TYPE ST_Initialisierungsroutine :
STRUCT

    MGMT_Parameter : ST_FB_MGMT_Parameter;
	Netze_Parameter :ST_Netze_Parameter;

	Anlage_BSp_Parameter	: ST_BSp_Parameter;
	Anlage_Bel_Parameter	: ST_Bel_Parameter;
	Anlage_BHKW_921_Parameter	: ST_BHKW_Parameter;
	Anlage_BHKW_922_Parameter	: ST_BHKW_Parameter;
	Anlage_BWK_Parameter	: ST_BWK_Parameter;
	Anlage_DLK_Parameter	: ST_DLK_Parameter;
	Anlage_HES_Parameter	: ST_HES_Parameter;
	Anlage_HO_Parameter		: ST_HO_Parameter;
	Anlage_LA_Parameter		: ST_LA_Parameter;
	Anlage_MVHW_Parameter	: ST_MV_JAVA_Parameter;
	Anlage_MVKW_Parameter	: ST_MV_MAFAC_GT_Parameter;
	Anlage_WP_946_Parameter		: ST_WP_Parameter;

	System_AFA_Parameter	: ST_System_AFA_Parameter;
	System_AKM_Parameter	: ST_System_AKM_Parameter;
	System_Bel_Parameter	: ST_System_Bel_Parameter;
	System_BHKW_Parameter	: ST_System_BHKW_Parameter;
	System_BSp_Parameter	: ST_System_BSp_Parameter;
	System_BSp_KueW_Parameter	: ST_System_BSp_KueW_Parameter;
	System_BSp_Verb_Parameter	: ST_System_BSp_Verb_Parameter;
	System_BWK_Parameter	: ST_System_BWK_Parameter;
	System_DLK_Parameter	: ST_System_DLK_Parameter;
	System_FBT_Parameter	: ST_System_FBT_Parameter;
	System_HES_Parameter	: ST_System_HES_Parameter;
	System_HOHW_Parameter	: ST_System_HOHW_Parameter;
	System_HOWW_Parameter	: ST_System_HOWW_Parameter;
	System_HS_Parameter		: ST_System_HS_Parameter;
	System_KKKW_Parameter	: ST_System_KKKW_Parameter;
	System_MVWW_Parameter	: ST_System_MVWW_Parameter;
	System_LA_Parameter		: ST_System_LA_Parameter;
	System_MVHW_Parameter	: ST_System_MVHW_Parameter;
	System_MVKW_Parameter	: ST_System_MVKW_Parameter;
	System_SHZ_Parameter	: ST_System_SHZ_Parameter;
	System_ThNTZ_Parameter	: ST_ThNTZ_Parameter;
	System_WDT_Parameter	: ST_System_WDT_Parameter;
	System_WT_HWW_Parameter	: ST_System_WT_HWW_Parameter;
	System_WP_946_Parameter		: ST_System_WP_Parameter;

	Fenster_Halle_OST_Parameter		: ST_Fenster_Parameter;
	Fenster_Halle_WEST_Parameter	: ST_Fenster_Parameter;


	Stellventil_100_Parameter	: ST_SV_Parameter;
	Stellventil_105_Parameter	:  ST_SV_Parameter;
	Stellventil_145_Parameter	:  ST_SV_Parameter;
	Stellventil_191_Parameter	: ST_SV_Parameter;
	Stellventil_205_Parameter	:  ST_SV_Parameter;
	Stellventil_215_Parameter	:  ST_SV_Parameter;
	Stellventil_235_Parameter	:  ST_SV_Parameter;
	Stellventil_245_Parameter	:  ST_SV_Parameter;
	Stellventil_251_Parameter	: ST_SV_Parameter;
	Stellventil_261_Parameter	: ST_SV_Parameter;
	Stellventil_300_Parameter	:  ST_SV_Parameter;
	Stellventil_315_Parameter	:  ST_SV_Parameter;
	Stellventil_321_Parameter	:  ST_SV_Parameter;
	Stellventil_322_Parameter	:  ST_SV_Parameter;
	Stellventil_331_Parameter	:  ST_SV_Parameter;
	Stellventil_361_Parameter	:  ST_SV_Parameter;
	Stellventil_423_Parameter	:  ST_SV_Parameter;
	Stellventil_424_Parameter	: ST_SV_Parameter;
	Stellventil_453_Parameter	: ST_SV_Parameter;
	Stellventil_454_Parameter	: ST_SV_Parameter;
	Stellventil_401_402_Parameter	: ST_SV_Parameter;
	Stellventil_403_404_Parameter	: ST_SV_Parameter;
	Stellventil_504_505_Parameter	:  ST_SV_Parameter;
	Stellventil_605_Parameter	: ST_SV_Parameter;

	Stellventil_146_Parameter	: ST_SV_Parameter;
	Stellventil_246_Parameter	:  ST_SV_Parameter;

	Pumpe_100_Parameter			: ST_PU_Parameter;
	Pumpe_105_Parameter			: ST_PU_Parameter;
	Pumpe_145_Parameter			: ST_PU_Parameter;
	Pumpe_191_Parameter			: ST_PU_Parameter;
	Pumpe_205_Parameter			: ST_PU_Parameter;
	Pumpe_215_Parameter			: ST_PU_Parameter;
	Pumpe_235_Parameter			: ST_PU_Parameter;
	Pumpe_245_Parameter			: ST_PU_Parameter;
	Pumpe_251_Parameter			: ST_PU_Parameter;
	Pumpe_261_Parameter			: ST_PU_Parameter;
	Pumpe_300_Parameter			: ST_PU_Parameter;
	Pumpe_315_Parameter			: ST_PU_Parameter;
	Pumpe_321_Parameter			: ST_PU_Parameter;
	Pumpe_322_Parameter			: ST_PU_Parameter;
	Pumpe_350_Parameter			: ST_PU_Parameter;
	Pumpe_361_Parameter			: ST_PU_Parameter;
	Pumpe_405_Parameter			: ST_PU_Parameter;
	Pumpe_425_Parameter			: ST_PU_Parameter;
	Pumpe_500_Parameter			: ST_PU_Parameter;
	Pumpe_600_Parameter			: ST_PU_Parameter;
	Pumpe_690_Parameter			: ST_PU_Schuetz_Parameter;
	Pumpe_710_Parameter			: ST_PU_Schuetz_Parameter;
	Pumpe_716_Parameter			: ST_PU_Schuetz_Parameter;
	Pumpe_720_Parameter			: ST_PU_Schuetz_Parameter;
	Pumpe_726_Parameter			: ST_PU_Schuetz_Parameter;
	Pumpe_760_Parameter			: ST_PU_Schuetz_Parameter;

	Regelventil_331_Parameter	:  ST_RV_Parameter;
	Regelventil_215_Parameter	:  ST_RV_Parameter;
	Regelventil_251_Parameter	:  ST_RV_Parameter;
	Regelventil_261_Parameter	:  ST_RV_Parameter;
	Regelventil_321_Parameter	:  ST_RV_Parameter;
	Regelventil_322_Parameter	:  ST_RV_Parameter;
	Regelventil_350_Parameter	: ST_RV_Parameter;
	Regelventil_361_Parameter	:  ST_RV_Parameter;
	Regelventil_425_Parameter	: ST_RV_Parameter;
	Regelventil_500_Parameter	: ST_RV_Parameter;
	Regelventil_541_Parameter	:  ST_RV_Parameter;
	Regelventil_542_Parameter	: ST_RV_Parameter;
	Regelventil_543_Parameter	: ST_RV_Parameter;
	Regelventil_551_Parameter	: ST_RV_Parameter;
	Regelventil_552_Parameter	:  ST_RV_Parameter;
	Regelventil_553_Parameter	:  ST_RV_Parameter;
	Regelventil_561_Parameter	:  ST_RV_Parameter;
	Regelventil_562_Parameter	: ST_RV_Parameter;
	Regelventil_563_Parameter	: ST_RV_Parameter;
	Regelventil_571_Parameter	: ST_RV_Parameter;
	Regelventil_572_Parameter	: ST_RV_Parameter;
	Regelventil_573_Parameter	: ST_RV_Parameter;
	Regelventil_600_Parameter	: ST_RV_Parameter;
	Regelventil_640_Parameter	: ST_RV_Parameter;
	Regelventil_660_Parameter	: ST_RV_Parameter;



END_STRUCT
END_TYPE

(* stored: Version 1.1.0.1, ProductVersion 3.1.4024.9
   DUT ST_Initialisierungsroutine: Id {1b5c8048-5f7c-4e25-8c12-7c0a2a44180b} *)
